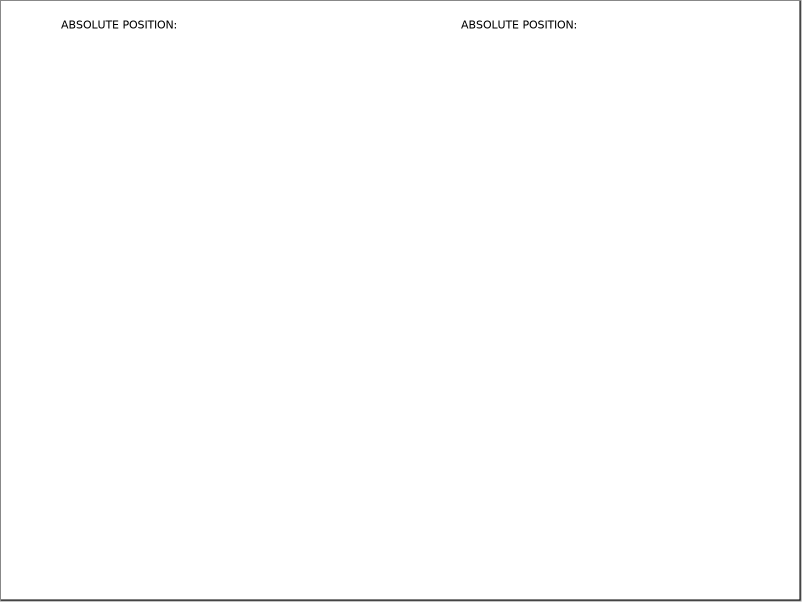
VISUALIZATION F11_Write_Digital_Output  // 802x602
    Rectangle (0,0 800x600)
    Label (10,10 170x30), "ABSOLUTE POSITION:"
    Label (410,10 170x30), "ABSOLUTE POSITION:"
END_VISUALIZATION

(* stored: Version 1.1.0.1, ProductVersion 3.1.4022.7
   Visu F11_Write_Digital_Output: Id {9cbc3fb0-82bf-4f31-b135-00cce6adc097} *)
